(* Logix 5000 project; controller Reto1_Fisico vendor 1 type 14 code 156 rev 30.11; software revision 30.00 *)

TASK MainTask (continuous, watchdog 500 ms) : MainProgram

MODULES
   Local : vendor 1 type 14 code 156 (Compact 0, rev 30.11)
      DigIN : 1769-IQ16 (Compact 4, rev 1.1, Input RPI 20 ms)
      DigOUT : vendor 1 type 7 code 86 (Compact 5, rev 2.1, Output RPI 20 ms)
END_MODULES

VAR_GLOBAL   (* controller tags *)
   Arranque_Fisico : ALIAS FOR Local:4:I.Data.1;   // Boton verde Fisico
   Contraer_D_E : ALIAS FOR Local:5:O.Data.5;   // Valvula para extender piston D.E. Fisico
   CTU_01 : COUNTER := (PRE := 1);   // ¿Hay cajas en banda 2?
   CTU_02 : COUNTER;   // Contador de caja bajando rampa final
   D_IN_1 : BOOL;   // Sensor 1 FactoryIO
   D_IN_2 : BOOL;   // Sensor 2 FactoryIO
   D_IN_3 : BOOL;   // Boton Stop FactoryIO
   D_IN_4 : BOOL;   // Boton Emergency Stop FactoryIO
   D_IN_5 : BOOL;   // Boton Start FactoryIO
   D_IN_6 : BOOL;   // Boton Reset FactoryIO
   D_IN_8 : BOOL;   // FactoryIO Running
   D_OUT_4 : BOOL;   // Banda 1 FactoryIO
   D_OUT_6 : BOOL;   // Compuerta FactoryIO
   Extender_D_E : ALIAS FOR Local:5:O.Data.4;   // Valvula para extender piston D.E. Fisico
   Extender_S_E : ALIAS FOR Local:5:O.Data.6;   // Valvula para extender piston S.E. Fisico
   F_OUT_1 : REAL;   // Banda 2 FactoryIO
   INT_OUT_0 : DINT;   // Display contador FactoryIO
   Motor_Fisico1 : ALIAS FOR Local:5:O.Data.0;   // Motor AC Fisico
   OSF01_OB : BOOL;   // Caja terminando de pasar por sensor 1
   OSF01_SB : BOOL;
   OSF02_OB : BOOL;   // ¿La caja ya bajo por la rampa final?
   OSF02_SB : BOOL;
   Stop_Fisico : ALIAS FOR Local:4:I.Data.0;   // Boton rojo Fisico
   Temp : BOOL;
   temp2 : BOOL;
   temp3 : BOOL;
   TIM_01 : TIMER := (PRE := 150);   // Caja ya paso por la compuerta
   TIM_02 : TIMER := (PRE := 150);   // Siguiente caja ya esta llegando a la compuerta
   TIM_03 : TIMER := (PRE := 1500);   // Diferencia Fisica vs FactoryIO
END_VAR

PROGRAM MainProgram   (* main routine MainRoutine *)

ROUTINE MainRoutine   (* ladder *)
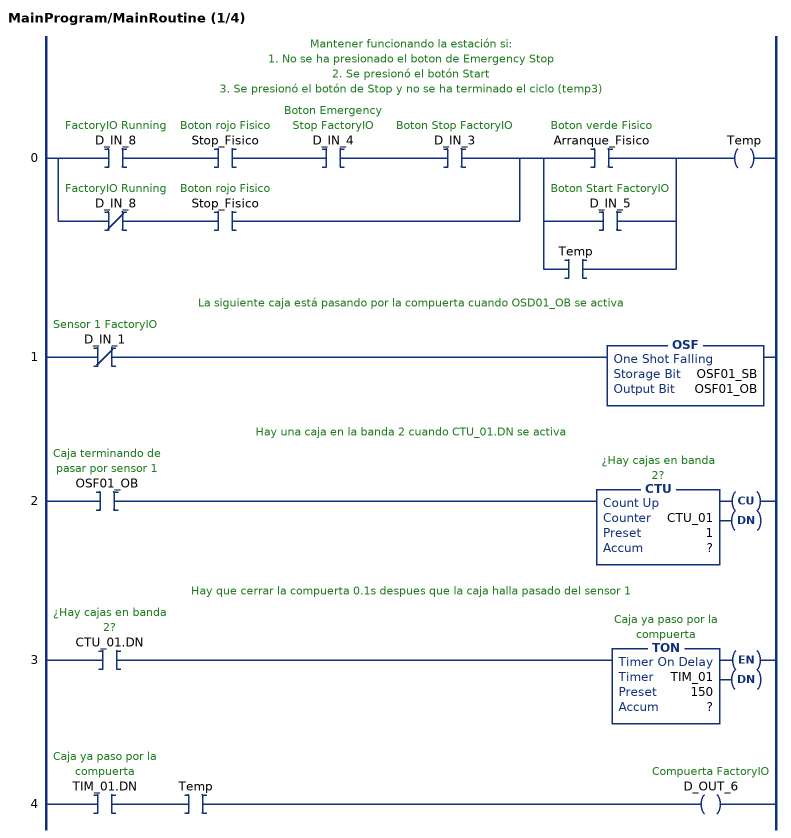
   // Mantener funcionando la estación si:
   // 1. No se ha presionado el boton de Emergency Stop
   // 2. Se presionó el botón Start
   // 3. Se presionó el botón de Stop y no se ha terminado el ciclo (temp3)
   0: [XIC(D_IN_8) XIC(Stop_Fisico) XIC(D_IN_4) XIC(D_IN_3) ,XIO(D_IN_8) XIC(Stop_Fisico) ][XIC(Arranque_Fisico) ,[XIC(D_IN_5) ,XIC(Temp) ] ]OTE(Temp);
   // La siguiente caja está pasando por la compuerta cuando OSD01_OB se activa
   1: XIO(D_IN_1)OSF(OSF01_SB,OSF01_OB);
   // Hay una caja en la banda 2 cuando CTU_01.DN se activa
   2: XIC(OSF01_OB)CTU(CTU_01,?,?);
   // Hay que cerrar la compuerta 0.1s despues que la caja halla pasado del sensor 1
   3: XIC(CTU_01.DN)TON(TIM_01,?,?);
   4: XIC(TIM_01.DN)XIC(Temp)OTE(D_OUT_6);
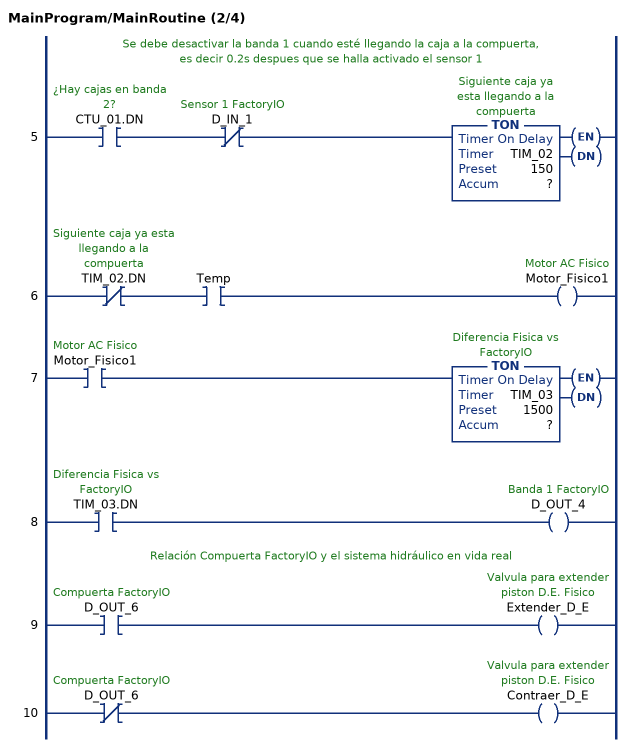
   // Se debe desactivar la banda 1 cuando esté llegando la caja a la compuerta,
   // es decir 0.2s despues que se halla activado el sensor 1
   5: XIC(CTU_01.DN)XIO(D_IN_1)TON(TIM_02,?,?);
   6: XIO(TIM_02.DN)XIC(Temp)OTE(Motor_Fisico1);
   7: XIC(Motor_Fisico1)TON(TIM_03,?,?);
   8: XIC(TIM_03.DN)OTE(D_OUT_4);
   // Relación Compuerta FactoryIO y el sistema hidráulico en vida real
   9: XIC(D_OUT_6)OTE(Extender_D_E);
   10: XIO(D_OUT_6)OTE(Contraer_D_E);
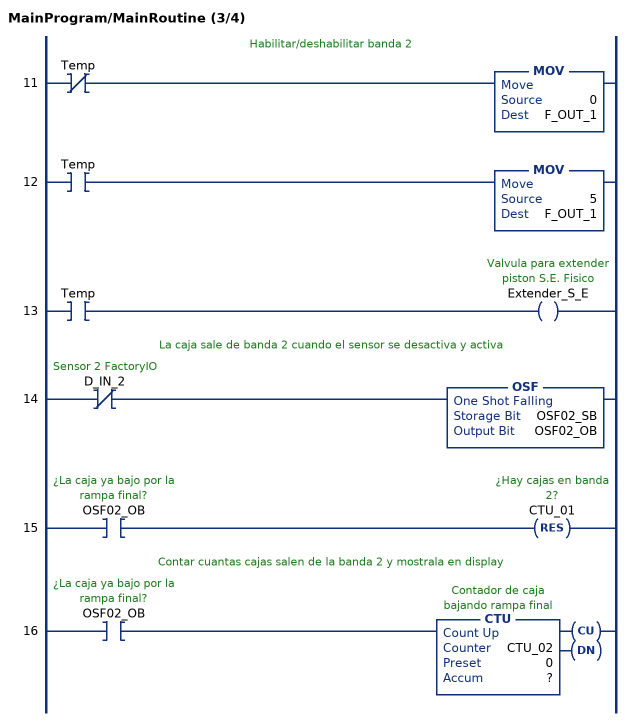
   // Habilitar/deshabilitar banda 2
   11: XIO(Temp)MOV(0,F_OUT_1);
   12: XIC(Temp)MOV(5,F_OUT_1);
   13: XIC(Temp)OTE(Extender_S_E);
   // La caja sale de banda 2 cuando el sensor se desactiva y activa
   14: XIO(D_IN_2)OSF(OSF02_SB,OSF02_OB);
   15: XIC(OSF02_OB)RES(CTU_01);
   // Contar cuantas cajas salen de la banda 2 y mostrala en display
   16: XIC(OSF02_OB)CTU(CTU_02,?,?);
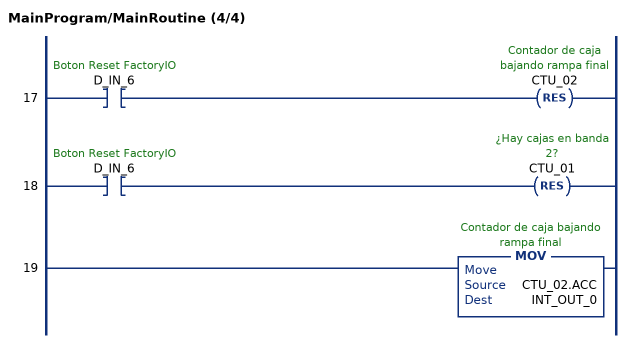
   17: XIC(D_IN_6)RES(CTU_02);
   18: XIC(D_IN_6)RES(CTU_01);
   19: MOV(CTU_02.ACC,INT_OUT_0);
END_ROUTINE
END_PROGRAM
